// TIA Portal V19 export
FUNCTION_BLOCK "LKinMAxisCtrlApcFr_Main"   // FB14, LAD
{ S7_Optimized_Access := 'TRUE' }
// stored: MemoryReserve 100, SetENOAutomatically false
   VAR_INPUT
      FirstCycle : Bool;
      Enable : Bool;
      StateSafetyActive : Bool := TRUE;
      StateInfeedInOperation : Bool;
      PowerAxisRobot { ExternalAccessible := 'False'; ExternalVisible := 'False'; ExternalWritable := 'False'} : Bool;
      Reset { ExternalAccessible := 'False'; ExternalVisible := 'False'; ExternalWritable := 'False'} : Bool;
      Home { ExternalAccessible := 'False'; ExternalVisible := 'False'; ExternalWritable := 'False'} : Bool;
      Data : "LKinMAxisCtrlApcFr_TypeDataParameters";
   END_VAR
   VAR_OUTPUT
      AxisPowered : Bool;
      AxisHomed : Bool;
      AxisError : Bool;
      KinematicError : Bool;
      KinematicInterrupted : Bool;
      AxisActualPosition : Array[1..6] of Real;
      KinematicActualPosition : Array[1..6] of Real;
      KinematicActualVelocity : Real;
   END_VAR
   VAR_IN_OUT
      AxisFB_Interface : Array[1.."LMAXISCTRLAPCFR_MAX_NUMBER_OF_AXES"] of "LMAxisCtrlApcFr_TypeInterface";
      Robot : TO_Kinematics;
   END_VAR
   VAR
      instLKinAxisCtrl_GroupPowered { S7_SetPoint := 'True'} : "LKinAxisCtrl_GroupPowered";
      instLKinAxisCtrl_GroupHomed { S7_SetPoint := 'True'} : "LKinAxisCtrl_GroupHomed";
      instLKinAxisCtrl_GroupError { S7_SetPoint := 'True'} : "LKinAxisCtrl_GroupError";
      "instLKinAxisCtrl_GroupPos&Velo" { S7_SetPoint := 'True'} : "LKinAxisCtrl_GroupPos&Velo";
      instLKinCtrl_GetKinematicsStatusWord { S7_SetPoint := 'True'} : "LKinCtrl_GetKinematicsStatusWord";
      instLKinAxisCtrlApcFr_CmdMAxisFB { S7_SetPoint := 'True'} : "LKinMAxisCtrlApcFr_CmdMAxisFB";
      instMC_RESET_Kinematic { S7_SetPoint := 'True'} : MC_RESET;
   END_VAR
BEGIN

REGION Network 1: Command Interface MAxisCtrlApcFr
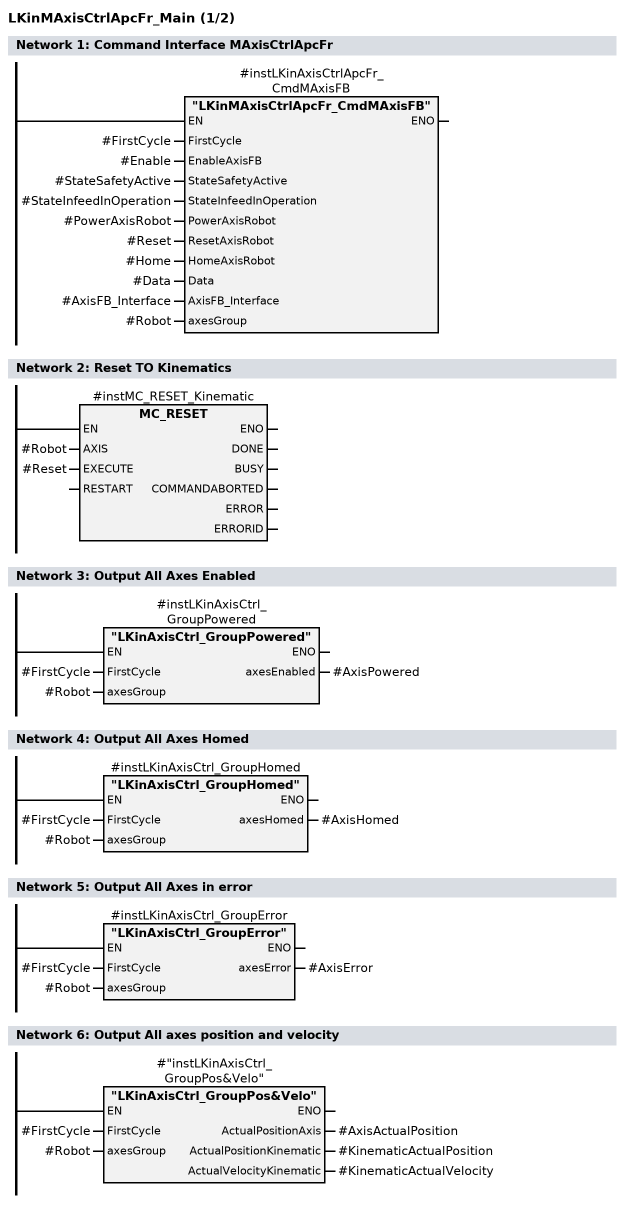
   RUNG wire#powerrail
      #instLKinAxisCtrlApcFr_CmdMAxisFB(FirstCycle := #FirstCycle, EnableAxisFB := #Enable, StateSafetyActive := #StateSafetyActive, StateInfeedInOperation := #StateInfeedInOperation, PowerAxisRobot := #PowerAxisRobot, ResetAxisRobot := #Reset, HomeAxisRobot := #Home, Data := #Data, AxisFB_Interface := #AxisFB_Interface, axesGroup := #Robot)
   END_RUNG
   // the same network as SCL:
   #instLKinAxisCtrlApcFr_CmdMAxisFB(FirstCycle := #FirstCycle,   // "LKinMAxisCtrlApcFr_CmdMAxisFB"
                           EnableAxisFB := #Enable,
                           StateSafetyActive := #StateSafetyActive,
                           StateInfeedInOperation := #StateInfeedInOperation,
                           PowerAxisRobot := #PowerAxisRobot,
                           ResetAxisRobot := #Reset,
                           HomeAxisRobot := #Home,
                           Data := #Data,
                           AxisFB_Interface := #AxisFB_Interface,
                           axesGroup := #Robot);
END_REGION

REGION Network 2: Reset TO Kinematics
   RUNG wire#powerrail
      #instMC_RESET_Kinematic.MC_RESET(Axis := #Robot, Execute := #Reset, Restart :=, Done =>, Busy =>, CommandAborted =>, Error =>, ErrorId =>)
   END_RUNG
   // the same network as SCL:
   #instMC_RESET_Kinematic(Axis := #Robot, Execute := #Reset);   // MC_RESET
END_REGION

REGION Network 3: Output All Axes Enabled
   RUNG wire#powerrail
      #instLKinAxisCtrl_GroupPowered(FirstCycle := #FirstCycle, axesGroup := #Robot, axesEnabled => #AxisPowered)
   END_RUNG
   // the same network as SCL:
   #instLKinAxisCtrl_GroupPowered(FirstCycle := #FirstCycle, axesGroup := #Robot, axesEnabled => #AxisPowered);   // "LKinAxisCtrl_GroupPowered"
END_REGION

REGION Network 4: Output All Axes Homed
   RUNG wire#powerrail
      #instLKinAxisCtrl_GroupHomed(FirstCycle := #FirstCycle, axesGroup := #Robot, axesHomed => #AxisHomed)
   END_RUNG
   // the same network as SCL:
   #instLKinAxisCtrl_GroupHomed(FirstCycle := #FirstCycle, axesGroup := #Robot, axesHomed => #AxisHomed);   // "LKinAxisCtrl_GroupHomed"
END_REGION

REGION Network 5: Output All Axes in error
   RUNG wire#powerrail
      #instLKinAxisCtrl_GroupError(FirstCycle := #FirstCycle, axesGroup := #Robot, axesError => #AxisError)
   END_RUNG
   // the same network as SCL:
   #instLKinAxisCtrl_GroupError(FirstCycle := #FirstCycle, axesGroup := #Robot, axesError => #AxisError);   // "LKinAxisCtrl_GroupError"
END_REGION

REGION Network 6: Output All axes position and velocity
   RUNG wire#powerrail
      #"instLKinAxisCtrl_GroupPos&Velo"(FirstCycle := #FirstCycle, axesGroup := #Robot, ActualPositionAxis => #AxisActualPosition, ActualPositionKinematic => #KinematicActualPosition, ActualVelocityKinematic => #KinematicActualVelocity)
   END_RUNG
   // the same network as SCL:
   #"instLKinAxisCtrl_GroupPos&Velo"(FirstCycle := #FirstCycle,   // "LKinAxisCtrl_GroupPos&Velo"
                           axesGroup := #Robot,
                           ActualPositionAxis => #AxisActualPosition,
                           ActualPositionKinematic => #KinematicActualPosition,
                           ActualVelocityKinematic => #KinematicActualVelocity);
END_REGION

REGION Network 7: Output Status TO Kinematic
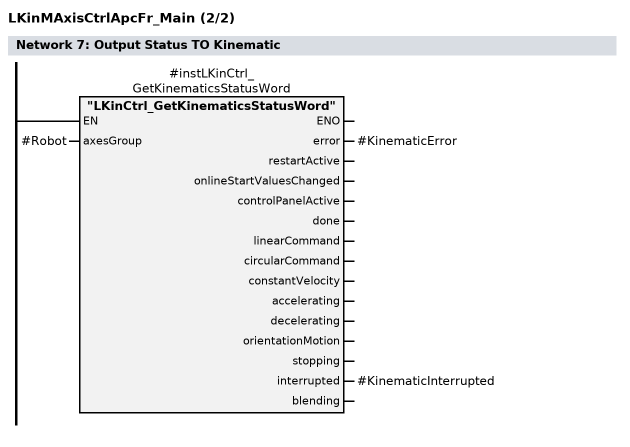
   RUNG wire#powerrail
      #instLKinCtrl_GetKinematicsStatusWord(axesGroup := #Robot, error => #KinematicError, restartActive =>, onlineStartValuesChanged =>, controlPanelActive =>, done =>, linearCommand =>, circularCommand =>, constantVelocity =>, accelerating =>, decelerating =>, orientationMotion =>, stopping =>, interrupted => #KinematicInterrupted, blending =>)
   END_RUNG
   // the same network as SCL:
   #instLKinCtrl_GetKinematicsStatusWord(axesGroup := #Robot,   // "LKinCtrl_GetKinematicsStatusWord"
                           error => #KinematicError,
                           interrupted => #KinematicInterrupted);
END_REGION
END_FUNCTION_BLOCK
